// Mitsubishi GX Works2 project: Control with Time Function   PLC: FX3S
// Control with Time Function

PROGRAM MAIN
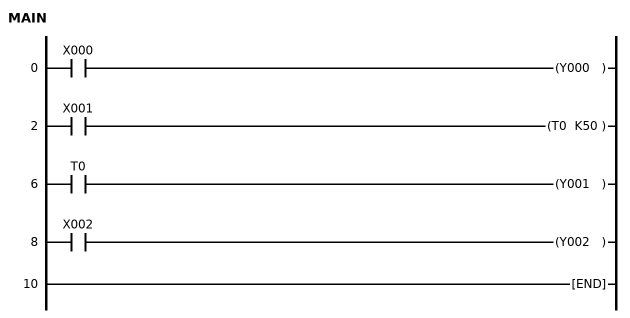
0     LD      X000
      OUT     Y000
2     LD      X001
      OUT     T0 K50
6     LD      T0
      OUT     Y001
8     LD      X002
      OUT     Y002
10    END
END_PROGRAM
